{attribute 'qualified_only'}
VAR_GLOBAL
	P1:BOOL; 	// Meldeleuchte weiss
	P2:BOOL;     // Meldeleuchte grün
	P3:BOOL;	//	Meldeleuchte rot
	Q1:BOOL;     // Motor Schnell (RL)
	Q2:BOOL;     // Motor Linkslauf
	Q3:BOOL;     // Motor Langsam (RL)
END_VAR

(* stored: Version 1.1.0.1, ProductVersion 3.1.4022.7
   GVL SimDA: Id {efa3d63a-96e1-4204-b1e7-9f3703bd4f03} *)
